FUNCTION Convert_TOD_TO_UDINT : BOOL
VAR_INPUT
	in : TOD;
	out : REFERENCE TO UDINT;
END_VAR
VAR
	converted : UDINT;
END_VAR

converted := TOD_TO_UDINT(in);

IF (UDINT_TO_TOD(converted) <> in) THEN
	RETURN;
END_IF

out := converted;
Convert_TOD_TO_UDINT := TRUE;

END_FUNCTION

(* stored: Version 1.1.0.1, ProductVersion 3.1.4024.12
   POU Convert_TOD_TO_UDINT: Id {2baf4923-3cab-46f7-8377-a4df670fa551}, SpecialFunc None *)
